# EPICS substitutions: iocBoot/ioc13Keithley3/pid_slow.substitutions
file "$(STD)/stdApp/Db/pid_control.db"
{
pattern
{P,            PID,       INP,           OUT,    LOPR,  HOPR,  DRVL,  DRVH,  PREC,   KP,  KI,   KD,  SCAN}
{13Keithley3:, PID1,  DMM1Ch1_calc.VAL, DAC1_4,   0,    100,     0,    5,     3,     0.2,  3.,   0.,  ".1 second"}
}
